// TIA Portal V19 export
DATA_BLOCK "InstFrequency"   // DB2
TITLE = InstFrequncy
{ DB_Accessible_From_OPC_UA := 'FALSE' }
// IDB Frequency
// stored: AssignedProDiagFB LiftProDiagFB, DBAccessibleFromOPCUA false, InstanceOfName Frequency, InstanceOfType FB
"Frequency"
   // VAR_INPUT
   //    frequency { ExternalAccessible := 'False'; ExternalVisible := 'False'; ExternalWritable := 'False'} : Real;
   // END_VAR
   // VAR_OUTPUT
   //    clock { ExternalAccessible := 'False'; ExternalVisible := 'False'; ExternalWritable := 'False'} : Bool;
   //    countdown { ExternalAccessible := 'False'; ExternalVisible := 'False'; ExternalWritable := 'False'} : Time;
   //    error { ExternalAccessible := 'False'; ExternalVisible := 'False'; ExternalWritable := 'False'} : Bool;
   //    status { ExternalAccessible := 'False'; ExternalVisible := 'False'; ExternalWritable := 'False'} : Word;
   // END_VAR
   // VAR
   //    instTofTimeOn { ExternalAccessible := 'False'; ExternalVisible := 'False'; ExternalWritable := 'False'; S7_SetPoint := 'True'} : TOF_TIME;
   //    instTofTimeOff { ExternalAccessible := 'False'; ExternalVisible := 'False'; ExternalWritable := 'False'; S7_SetPoint := 'True'} : TOF_TIME;
   //    statFrequencyMem { ExternalAccessible := 'False'; ExternalVisible := 'False'; ExternalWritable := 'False'} : Real;
   //    statTimeBase { ExternalAccessible := 'False'; ExternalVisible := 'False'; ExternalWritable := 'False'} : Time;
   // END_VAR
BEGIN
END_DATA_BLOCK
